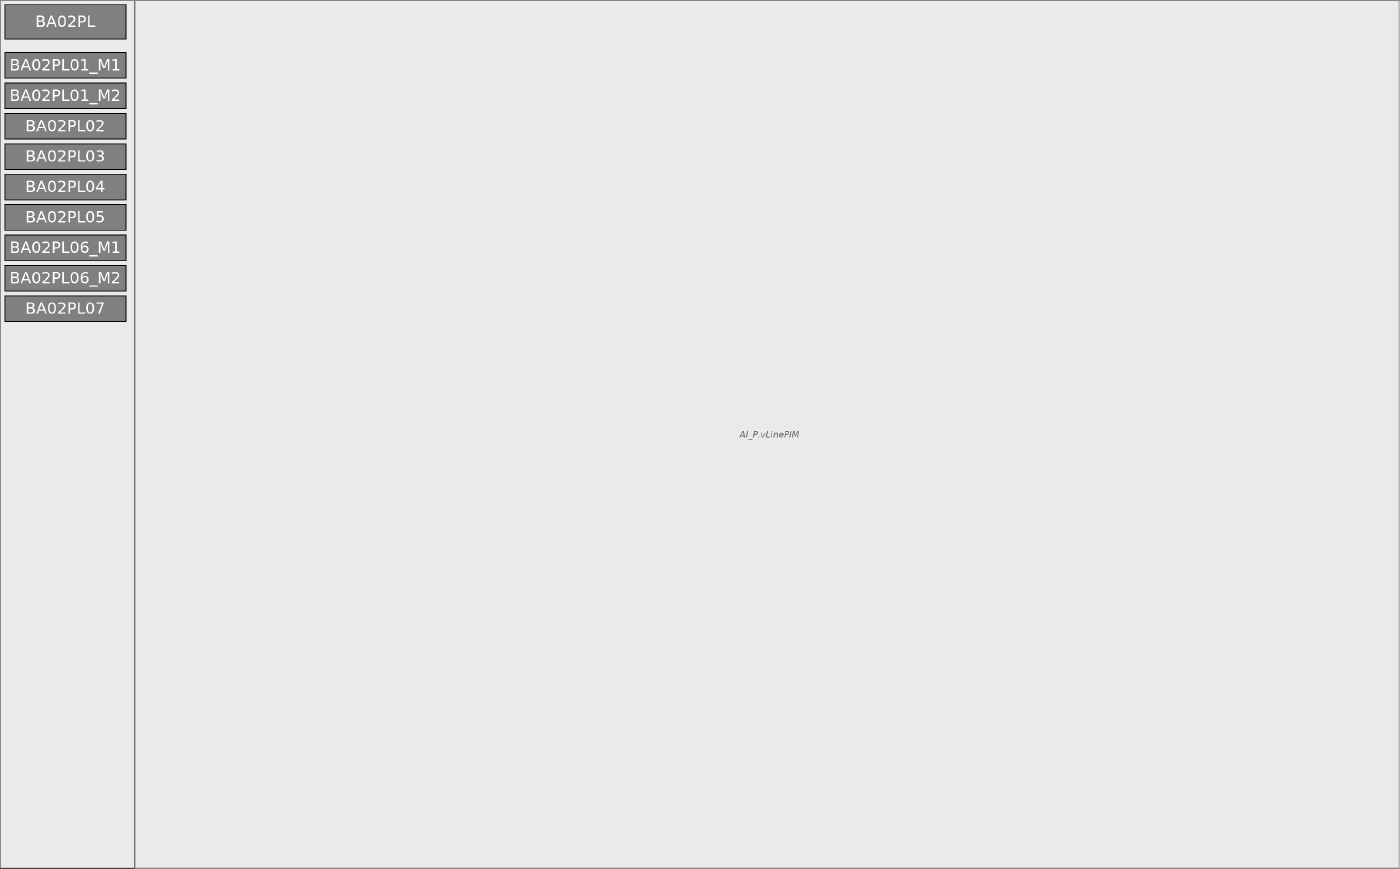
VISUALIZATION HomeVisuBA02PL  // 1610x1000
    Rectangle (0,0 155x1000)
    Frame (155,0 1460x1000)
        shows AI_P.vLinePIM(fbPIM := MAIN.stLine_BA02PL.fbLine)
        shows AI_P.vStationPIM(fbPIM := MAIN.fb_Filler_A_Machine.fbPIM)
        shows AI_P.vStationPIM(fbPIM := MAIN.fb_Cork_Machine.fbPIM)
        shows AI_P.vStationPIM(fbPIM := MAIN.fb_1_SonicTech_SonictechUSW.fbPIM)
        shows AI_P.vStationPIM(fbPIM := MAIN.fb_Filler_B_Machine.fbPIM)
        shows AI_P.vStationPIM(fbPIM := MAIN.fb_2_SonicTech_SonictechUSW.fbPIM)
        shows AI_P.vStationPIM(fbPIM := MAIN.fb_UnderPressure_Tester_Machine.fbPIM)
        shows AI_P.vStationPIM(fbPIM := MAIN.fb_Sticker_Machine.fbPIM)
        shows AI_P.vStationPIM(fbPIM := MAIN.fb_Laser_Machine.fbPIM)
        shows AI_P.vStationPIM(fbPIM := MAIN.fbWeighingTunel.fbTableControl.fbPIM)
        shows AircomLibrary.vStationPIM(fbPIM := MAIN.fbS19_2_EOL3.fbPIM)
        shows AircomLibrary.vStationPIM(fbPIM := MAIN.fbS20_AssemblyPost.fbPIM)
        shows AircomLibrary.vStationPIM(fbPIM := MAIN.fbS21_DetectionTunel.fbPIM)
        shows AircomLibrary.vStationPIM(fbPIM := MAIN.fbS22_SetPackingStation.fbPIM)
        p2766960713: GVL.fbSqlCore
        p2683556743: GVL.stLJ20_DTL_WorkParams
        p3043078949: MAIN.fbLL19_1_EOL3
        p1709583229: GVL.stLL19_EOL_Settings_I
        p2719655782: MAIN.fbLL19_2_EOL3
        p3094409976: GVL.stLL19_EOL_Settings_II
        p74549115: 'Left chamber'
        p3369830373: 'Right chamber'
        p3445515547: MAIN.fbLS06
        p3589162504: GVL_IO.stLS01_HoseCutter
        p458721708: MAIN.fbLS01_HoseCutter
        p3390713232: MAIN.fbLS04_1_Station
        p1393785898: MAIN.fbLS04_2_Station
        p3419948967: MAIN.fbLS05_1_Station
        p1389434397: MAIN.fbLS05_2_Station
        p422258626: MAIN.fbLS04_1_Crimper
        p417943029: MAIN.fbLS05_1_Crimper
        p2149742200: MAIN.fbLS04_2_Crimper
        p2178948175: MAIN.fbLS05_2_Crimper
        p180551898: MAIN.fbS03
        p2110009420: MAIN.fbLS02_InsertAssy
        p2404496545: MAIN.fbLS02_Station
        p4166419511: MAIN.fbLS03_Station
        p1449093633: MAIN.fbLS06_V2
        p898092448: GVL.Hose_Tester_Params_V2
        p589997586: GVL.Hose_Tester_Params_V2.iPickedHose
        p1762866656: MAIN.fbS03
        p504628598: MAIN.fbLS02_InsertAssy
        p1957019379: MAIN.fbLS06_V2
        p1712759876: GVL.Hose_Tester_Params_V2
        p3689475492: GVL.Hose_Tester_Params_V2.iPickedHose
        p1628323955: MAIN.fbS21_DetectionTunel.fbPIM
        p2913222893: MAIN.fbS22_SetPackingStation.fbPIM
    Rectangle (5,5 140x40), "BA02PL"
        OnMouseDown: FrameSelectionChange Selection=SelectedFrame=cd818c81-a6c5-4ab8-9515-1ee8055884ac, GlobSel=AssignType=Directly, SelType=Locally
    Rectangle (5,60 140x30), "BA02PL01_M1"
        OnMouseDown: FrameSelectionChange Selection=SelectedFrame=cd818c81-a6c5-4ab8-9515-1ee8055884ac, Selection=1, GlobSel=AssignType=Directly, SelType=Locally
    Rectangle (5,165 140x30), "BA02PL03"
        OnMouseDown: FrameSelectionChange Selection=SelectedFrame=cd818c81-a6c5-4ab8-9515-1ee8055884ac, Selection=4, GlobSel=AssignType=Directly, SelType=Locally
    Rectangle (5,95 140x30), "BA02PL01_M2"
        OnMouseDown: FrameSelectionChange Selection=SelectedFrame=cd818c81-a6c5-4ab8-9515-1ee8055884ac, Selection=2, GlobSel=AssignType=Directly, SelType=Locally
    Rectangle (5,130 140x30), "BA02PL02"
        OnMouseDown: FrameSelectionChange Selection=SelectedFrame=cd818c81-a6c5-4ab8-9515-1ee8055884ac, Selection=3, GlobSel=AssignType=Directly, SelType=Locally
    Rectangle (5,200 140x30), "BA02PL04"
        OnMouseDown: FrameSelectionChange Selection=SelectedFrame=cd818c81-a6c5-4ab8-9515-1ee8055884ac, Selection=5, GlobSel=AssignType=Directly, SelType=Locally
    Rectangle (5,235 140x30), "BA02PL05"
        OnMouseDown: FrameSelectionChange Selection=SelectedFrame=cd818c81-a6c5-4ab8-9515-1ee8055884ac, Selection=6, GlobSel=AssignType=Directly, SelType=Locally
    Rectangle (5,305 140x30), "BA02PL06_M2"
        OnMouseDown: FrameSelectionChange Selection=SelectedFrame=cd818c81-a6c5-4ab8-9515-1ee8055884ac, Selection=8, GlobSel=AssignType=Directly, SelType=Locally
    Rectangle (5,270 140x30), "BA02PL06_M1"
        OnMouseDown: FrameSelectionChange Selection=SelectedFrame=cd818c81-a6c5-4ab8-9515-1ee8055884ac, Selection=7, GlobSel=AssignType=Directly, SelType=Locally
    Rectangle (5,340 140x30), "BA02PL07"
        OnMouseDown: FrameSelectionChange Selection=SelectedFrame=cd818c81-a6c5-4ab8-9515-1ee8055884ac, Selection=9, GlobSel=AssignType=Directly, SelType=Locally
END_VISUALIZATION

(* stored: Version 1.1.0.1, ProductVersion 3.1.4024.16
   Visu HomeVisuBA02PL: Id {cf9ee581-cf1b-48bc-bdce-76b7c0b1c84e} *)
